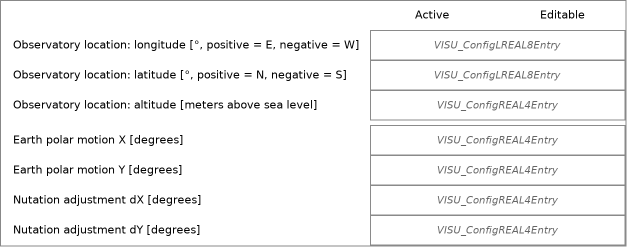
VISUALIZATION VISU_AxesConfig_Location  // 627x247
VAR_IN_OUT
    active : AxesLocationConfig;
    editable : AxesLocationConfig;
END_VAR
    Label (370,5 125x20), "Active"
    Label (500,5 125x20), "Editable"
    Label (10,30 360x30), "Observatory location: longitude [°, positive = E, negative = W]"
    Frame (370,30 255x30)
        shows VISU_ConfigLREAL8Entry(active := active.longitude, editable := editable.longitude)
    Frame (370,60 255x30)
        shows VISU_ConfigLREAL8Entry(active := active.latitude, editable := editable.latitude)
    Label (10,60 360x30), "Observatory location: latitude [°, positive = N, negative = S]"
    Label (10,90 360x30), "Observatory location: altitude [meters above sea level]"
    Frame (370,90 255x30)
        shows VISU_ConfigREAL4Entry(active := active.height, editable := editable.height)
    Label (10,125 360x30), "Earth polar motion X [degrees]"
    Frame (370,125 255x30)
        shows VISU_ConfigREAL4Entry(active := active.polarMotionX, editable := editable.polarMotionX)
    Label (10,155 360x30), "Earth polar motion Y [degrees]"
    Frame (370,155 255x30)
        shows VISU_ConfigREAL4Entry(active := active.polarMotionY, editable := editable.polarMotionY)
    Frame (370,185 255x30)
        shows VISU_ConfigREAL4Entry(active := active.nutationDx, editable := editable.nutationDx)
    Label (10,185 360x30), "Nutation adjustment dX [degrees]"
    Label (10,215 360x30), "Nutation adjustment dY [degrees]"
    Frame (370,215 255x30)
        shows VISU_ConfigREAL4Entry(active := active.nutationDy, editable := editable.nutationDy)
END_VISUALIZATION

(* stored: Version 1.1.0.1, ProductVersion 3.1.4019.2
   Visu VISU_AxesConfig_Location: Id {f1d0c650-2e3b-4a36-bb69-1735495c0f82} *)
